TYPE CardboardMaterial :
STRUCT
	foldType : (FLAT, CORNER, COVER);
	foldPos1 : REAL;
	foldPos2 : REAL;
END_STRUCT
END_TYPE

(* stored: Version 1.1.0.1, ProductVersion 3.1.4024.11
   DUT CardboardMaterial: Id {f4eae4b3-bd31-4fd7-9db3-f96f03e355e4} *)
